// Mitsubishi GX Works2 project: 시퀀스 예제 1_2   PLC: Q03UDV

PROGRAM MAIN
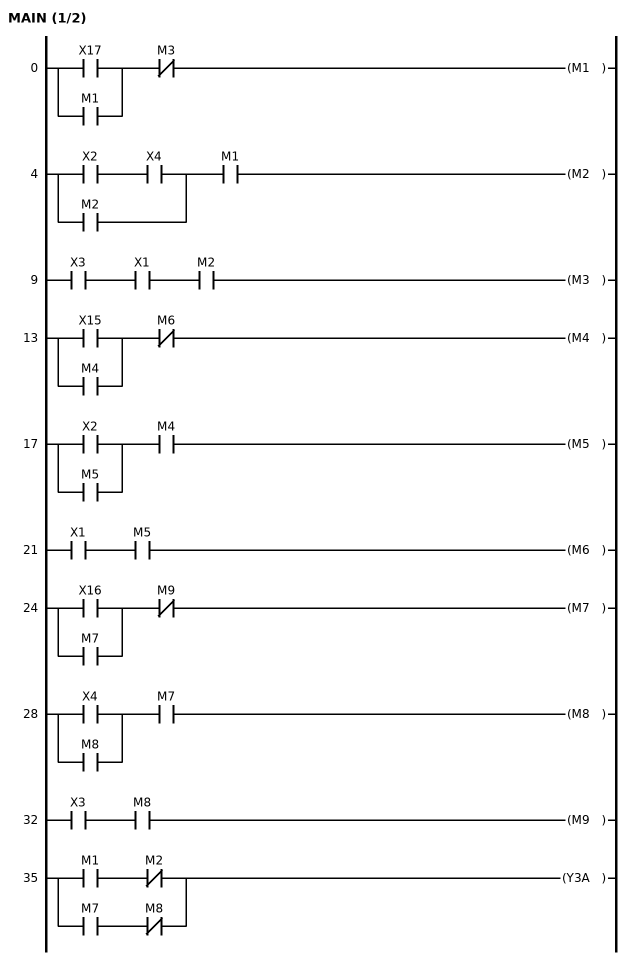
0     LD      X17
      OR      M1
      ANI     M3
      OUT     M1
4     LD      X2
      AND     X4
      OR      M2
      AND     M1
      OUT     M2
9     LD      X3
      AND     X1
      AND     M2
      OUT     M3
13    LD      X15
      OR      M4
      ANI     M6
      OUT     M4
17    LD      X2
      OR      M5
      AND     M4
      OUT     M5
21    LD      X1
      AND     M5
      OUT     M6
24    LD      X16
      OR      M7
      ANI     M9
      OUT     M7
28    LD      X4
      OR      M8
      AND     M7
      OUT     M8
32    LD      X3
      AND     M8
      OUT     M9
35    LD      M1
      ANI     M2
      LD      M7
      ANI     M8
      ORB
      OUT     Y3A
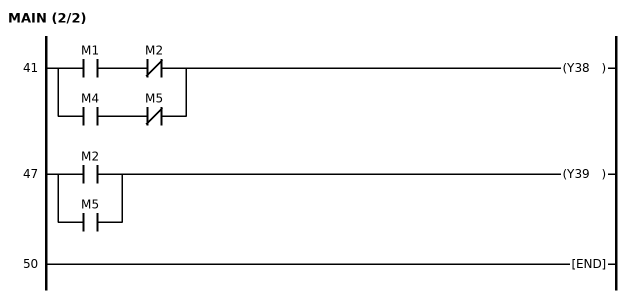
41    LD      M1
      ANI     M2
      LD      M4
      ANI     M5
      ORB
      OUT     Y38
47    LD      M2
      OR      M5
      OUT     Y39
50    END
END_PROGRAM
